FUNCTION_BLOCK FB_System_SHZ_Ablaufsteuerung
VAR_IN_OUT
	Zustand			: ST_System_SHZ_Zustand;
	Stellwert			: ST_System_SHZ_Stellwert;
	Steuerung			: ST_System_SHZ_Steuerung;
END_VAR
VAR_INPUT
	Zustand_Pumpe			: ST_PU_Zustand;
	Zustand_Regelventil		: ST_RV_Zustand;
END_VAR
VAR_OUTPUT
END_VAR
VAR
END_VAR

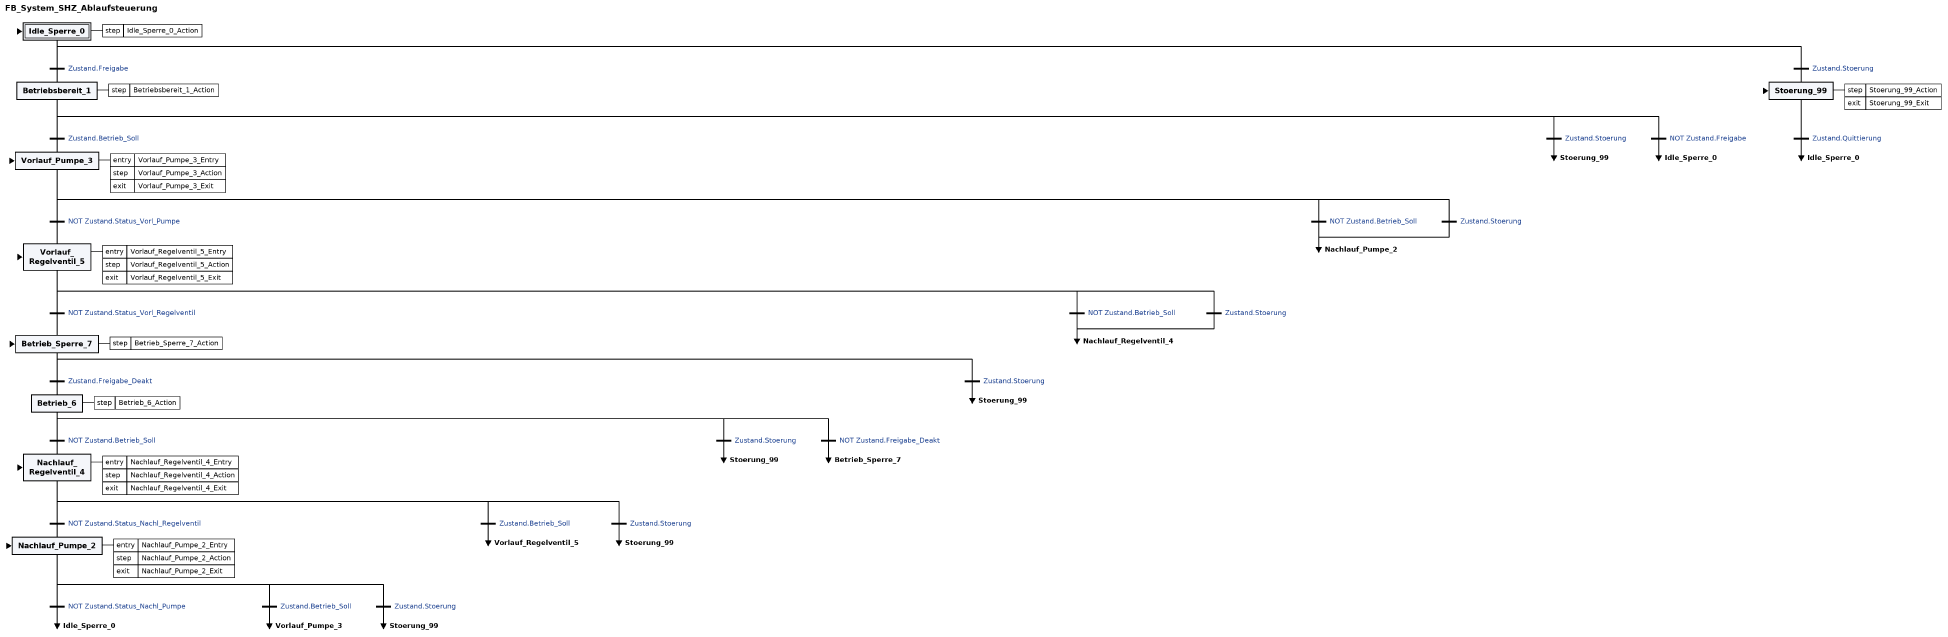
INITIAL_STEP Idle_Sperre_0:
    Idle_Sperre_0_Action(N);  // step action
END_STEP
TRANSITION FROM Idle_Sperre_0 TO Betriebsbereit_1
    := Zustand.Freigabe;
END_TRANSITION
TRANSITION FROM Idle_Sperre_0 TO Stoerung_99
    := Zustand.Stoerung;
END_TRANSITION
STEP Stoerung_99:
    Stoerung_99_Action(N);  // step action
    Stoerung_99_Exit(P0);  // exit action
END_STEP
TRANSITION FROM Stoerung_99 TO Idle_Sperre_0
    := Zustand.Quittierung;
END_TRANSITION
STEP Betriebsbereit_1:
    Betriebsbereit_1_Action(N);  // step action
END_STEP
TRANSITION FROM Betriebsbereit_1 TO Vorlauf_Pumpe_3
    := Zustand.Betrieb_Soll;
END_TRANSITION
TRANSITION FROM Betriebsbereit_1 TO Stoerung_99
    := Zustand.Stoerung;
END_TRANSITION
TRANSITION FROM Betriebsbereit_1 TO Idle_Sperre_0
    := NOT Zustand.Freigabe;
END_TRANSITION
STEP Vorlauf_Pumpe_3:
    Vorlauf_Pumpe_3_Entry(P1);  // entry action
    Vorlauf_Pumpe_3_Action(N);  // step action
    Vorlauf_Pumpe_3_Exit(P0);  // exit action
END_STEP
TRANSITION FROM Vorlauf_Pumpe_3 TO Vorlauf_Regelventil_5
    := NOT Zustand.Status_Vorl_Pumpe;
END_TRANSITION
TRANSITION FROM Vorlauf_Pumpe_3 TO Nachlauf_Pumpe_2
    := NOT Zustand.Betrieb_Soll;
END_TRANSITION
TRANSITION FROM Vorlauf_Pumpe_3 TO Nachlauf_Pumpe_2
    := Zustand.Stoerung;
END_TRANSITION
STEP Vorlauf_Regelventil_5:
    Vorlauf_Regelventil_5_Entry(P1);  // entry action
    Vorlauf_Regelventil_5_Action(N);  // step action
    Vorlauf_Regelventil_5_Exit(P0);  // exit action
END_STEP
TRANSITION FROM Vorlauf_Regelventil_5 TO Betrieb_Sperre_7
    := NOT Zustand.Status_Vorl_Regelventil;
END_TRANSITION
TRANSITION FROM Vorlauf_Regelventil_5 TO Nachlauf_Regelventil_4
    := NOT Zustand.Betrieb_Soll;
END_TRANSITION
TRANSITION FROM Vorlauf_Regelventil_5 TO Nachlauf_Regelventil_4
    := Zustand.Stoerung;
END_TRANSITION
STEP Betrieb_Sperre_7:
    Betrieb_Sperre_7_Action(N);  // step action
END_STEP
TRANSITION FROM Betrieb_Sperre_7 TO Betrieb_6
    := Zustand.Freigabe_Deakt;
END_TRANSITION
TRANSITION FROM Betrieb_Sperre_7 TO Stoerung_99
    := Zustand.Stoerung;
END_TRANSITION
STEP Betrieb_6:
    Betrieb_6_Action(N);  // step action
END_STEP
TRANSITION FROM Betrieb_6 TO Nachlauf_Regelventil_4
    := NOT Zustand.Betrieb_Soll;
END_TRANSITION
TRANSITION FROM Betrieb_6 TO Stoerung_99
    := Zustand.Stoerung;
END_TRANSITION
TRANSITION FROM Betrieb_6 TO Betrieb_Sperre_7
    := NOT Zustand.Freigabe_Deakt;
END_TRANSITION
STEP Nachlauf_Regelventil_4:
    Nachlauf_Regelventil_4_Entry(P1);  // entry action
    Nachlauf_Regelventil_4_Action(N);  // step action
    Nachlauf_Regelventil_4_Exit(P0);  // exit action
END_STEP
TRANSITION FROM Nachlauf_Regelventil_4 TO Nachlauf_Pumpe_2
    := NOT Zustand.Status_Nachl_Regelventil;
END_TRANSITION
TRANSITION FROM Nachlauf_Regelventil_4 TO Vorlauf_Regelventil_5
    := Zustand.Betrieb_Soll;
END_TRANSITION
TRANSITION FROM Nachlauf_Regelventil_4 TO Stoerung_99
    := Zustand.Stoerung;
END_TRANSITION
STEP Nachlauf_Pumpe_2:
    Nachlauf_Pumpe_2_Entry(P1);  // entry action
    Nachlauf_Pumpe_2_Action(N);  // step action
    Nachlauf_Pumpe_2_Exit(P0);  // exit action
END_STEP
TRANSITION FROM Nachlauf_Pumpe_2 TO Idle_Sperre_0
    := NOT Zustand.Status_Nachl_Pumpe;
END_TRANSITION
TRANSITION FROM Nachlauf_Pumpe_2 TO Vorlauf_Pumpe_3
    := Zustand.Betrieb_Soll;
END_TRANSITION
TRANSITION FROM Nachlauf_Pumpe_2 TO Stoerung_99
    := Zustand.Stoerung;
END_TRANSITION

ACTION Betrieb_6_Action:
(* Stellwert setzen *)
Stellwert.Anford_Pumpe		:= TRUE;
Stellwert.Anford_Regelventil		:= TRUE;

(* Zustand setzen *)
Zustand.Betrieb				:= TRUE;
Zustand.Status				:= E_System_SHZ_Zustand_Status_Betrieb;
END_ACTION

ACTION Betrieb_Sperre_7_Action:
(* Stellwert setzen *)
Stellwert.Anford_Pumpe		:= TRUE;
Stellwert.Anford_Regelventil		:= TRUE;

(* Zustand setzen *)
Zustand.Betrieb				:= TRUE;
Zustand.Status				:= E_System_SHZ_Zustand_Status_Betrieb_Sperre;
END_ACTION

ACTION Betriebsbereit_1_Action:
(* Stellwert setzen *)
Stellwert.Anford_Pumpe	:= FALSE;
Stellwert.Anford_Regelventil	:= FALSE;

(* Zustand setzen *)
Zustand.Betrieb			:= FALSE;
Zustand.Status			:= E_System_SHZ_Zustand_Status_Betriebsbereit;
Zustand.Regelung_Modus 	:= E_System_SHZ_Regelung_Modus_Automatik;
END_ACTION

ACTION Idle_Sperre_0_Action:
(* Stellwert setzen *)
Stellwert.Anford_Pumpe	:= FALSE;
Stellwert.Anford_Regelventil	:= FALSE;

(* Zustand setzen *)
Zustand.Betrieb			:= FALSE;
Zustand.Status			:= E_System_SHZ_Zustand_Status_Idle_Sperre;

(* Quittierungszustand auf False setzen, damit das System bei einer erneuten Störung nicht direkt wieder angeschaltet wird *)
Steuerung.Quittierung	:= FALSE;
END_ACTION

ACTION Nachlauf_Pumpe_2_Action:
(* Stellwert setzen *)
Stellwert.Anford_Pumpe		:= FALSE;
Stellwert.Anford_Regelventil		:= FALSE;

(* Zustand setzen *)
Zustand.Betrieb				:= FALSE;
Zustand.Status				:= E_System_SHZ_Zustand_Status_Nachl_Pumpe;
Zustand.Status_Nachl_Pumpe	:= Zustand_Pumpe.Betrieb OR Zustand_Pumpe.Status_Nachl;
END_ACTION

ACTION Nachlauf_Pumpe_2_Entry:
Zustand.Status_Nachl_Pumpe	:= TRUE;
END_ACTION

ACTION Nachlauf_Pumpe_2_Exit:
Zustand.Status_Nachl_Pumpe	:= FALSE;
END_ACTION

ACTION Nachlauf_Regelventil_4_Action:
(* Stellwert setzen *)
Stellwert.Anford_Pumpe		:= TRUE;
Stellwert.Anford_Regelventil		:= FALSE;

(* Zustand setzen *)
Zustand.Betrieb					:= FALSE;
Zustand.Status					:= E_System_SHZ_Zustand_Status_Nachl_Regelventil;
Zustand.Status_Nachl_Regelventil	:= Zustand_Regelventil.Betrieb OR Zustand_Regelventil.Status_Nachl;
END_ACTION

ACTION Nachlauf_Regelventil_4_Entry:
Zustand.Status_Nachl_Regelventil		:= TRUE;
END_ACTION

ACTION Nachlauf_Regelventil_4_Exit:
Zustand.Status_Nachl_Regelventil		:= FALSE;
END_ACTION

ACTION Stoerung_99_Action:
(* Stellwert setzen *)
Stellwert.Anford_Pumpe	:= FALSE;
Stellwert.Anford_Regelventil	:= FALSE;

(* Zustand setzen *)
Zustand.Betrieb			:= FALSE;
Zustand.Stoerung			:= TRUE;
Zustand.Status			:= E_System_SHZ_Zustand_Status_Stoerung;
END_ACTION

ACTION Stoerung_99_Exit:
Zustand.Stoerung	:= FALSE;
END_ACTION

ACTION Vorlauf_Pumpe_3_Action:
(* Stellwert setzen *)
Stellwert.Anford_Pumpe		:= TRUE;
Stellwert.Anford_Regelventil		:= FALSE;

(* Zustand setzen *)
Zustand.Betrieb				:= FALSE;
Zustand.Status				:= E_System_SHZ_Zustand_Status_Vorl_Pumpe;
Zustand.Status_Vorl_Pumpe	:= NOT(Zustand_Pumpe.Betrieb AND NOT Zustand_Pumpe.Status_Vorl);
END_ACTION

ACTION Vorlauf_Pumpe_3_Entry:
Zustand.Status_Vorl_Pumpe	:= TRUE;
END_ACTION

ACTION Vorlauf_Pumpe_3_Exit:
Zustand.Status_Vorl_Pumpe	:= FALSE;
END_ACTION

ACTION Vorlauf_Regelventil_5_Action:
(* Stellwert setzen *)
Stellwert.Anford_Pumpe		:= TRUE;
Stellwert.Anford_Regelventil		:= TRUE;

(* Zustand setzen *)
Zustand.Betrieb				:= FALSE;
Zustand.Status				:= E_System_SHZ_Zustand_Status_Vorl_Regelventil;
Zustand.Status_Vorl_Regelventil	:= NOT(Zustand_Regelventil.Betrieb AND NOT Zustand_Regelventil.Status_Vorl);
END_ACTION

ACTION Vorlauf_Regelventil_5_Entry:
Zustand.Status_Vorl_Regelventil	:= TRUE;
END_ACTION

ACTION Vorlauf_Regelventil_5_Exit:
Zustand.Status_Vorl_Regelventil		:= FALSE;
END_ACTION

END_FUNCTION_BLOCK

(* stored: Version 1.1.0.1, ProductVersion 3.1.4024.9
   POU FB_System_SHZ_Ablaufsteuerung: Id {5915c67f-150f-427c-b237-3796e584b845}, SpecialFunc None
   Action Betrieb_6_Action: Id {49055838-9eef-49ac-9e0d-616e6ea9f503}
   Action Betrieb_Sperre_7_Action: Id {ab23cad0-659f-4d85-8c43-2c54acc0e2f8}
   Action Betriebsbereit_1_Action: Id {01a04b97-7466-44d0-b472-d8449c7ce603}
   Action Idle_Sperre_0_Action: Id {b5d17328-63c2-4503-ac46-5afb559e1e10}
   Action Nachlauf_Pumpe_2_Action: Id {b4819172-6e9a-4121-9e40-ed8b0e09dfa8}
   Action Nachlauf_Pumpe_2_Entry: Id {52694fc9-82a1-45f2-94c6-a16c00e1e73b}
   Action Nachlauf_Pumpe_2_Exit: Id {c7baf47a-d494-4861-8ed2-cb53849e3ab1}
   Action Nachlauf_Regelventil_4_Action: Id {387cc12c-8bcf-494f-9cd0-3cf3ce5902e1}
   Action Nachlauf_Regelventil_4_Entry: Id {57e5f472-8e68-46e7-8c2c-28ff67514e34}
   Action Nachlauf_Regelventil_4_Exit: Id {743eb972-ccb3-42d7-9557-7c0bebe4908c}
   Action Stoerung_99_Action: Id {3bcd2ab4-f67e-49b7-8bec-0ab46ad6c242}
   Action Stoerung_99_Exit: Id {8a72f4d7-71f5-42fd-a782-7eec2fbfc13d}
   Action Vorlauf_Pumpe_3_Action: Id {e6f0f5e2-ca35-4346-9c14-25873eeea0d4}
   Action Vorlauf_Pumpe_3_Entry: Id {3d56a3a7-c72b-4ec5-9ab9-881aa8b860de}
   Action Vorlauf_Pumpe_3_Exit: Id {555953bf-2dda-4af0-af03-9bd039a1a4b4}
   Action Vorlauf_Regelventil_5_Action: Id {68be5887-2f5a-4fc9-8cd8-915b1f5752be}
   Action Vorlauf_Regelventil_5_Entry: Id {406ab71b-a7f2-441a-bfca-ec4bbd955388}
   Action Vorlauf_Regelventil_5_Exit: Id {4f4663ab-276c-43ad-aa01-849ccc5e3cd8} *)
